TEXTLIST TL_E_CTRL_TRANSPORT
  0 = 'CMD_NULL'
  10 = 'CMD_INIT'
  11 = 'CMD_IDLE'
  20 = 'CMD_MOVER_ENABLE'
  21 = 'CMD_MOVER_DISABLE'
  22 = 'CMD_MOVER_HALT_CA'
  23 = 'CMD_MOVER_STOP'
  30 = 'CMD_GROUP_CLEAR'
  31 = 'CMD_GROUP_BUILD'
  32 = 'CMD_GROUP_ENABLE'
  33 = 'CMD_GROUP_STOP'
  40 = 'CMD_TRANSPORT_START'
  41 = 'CMD_TRANSPORT_RESTART'
   = ''
END_TEXTLIST

(* stored: Version 1.1.0.1
   TextList TL_E_CTRL_TRANSPORT: Id {159f6868-5098-4130-9487-0215047a5d64} *)
